// TIA Portal project "Sorting_Station_Project" (V16)
// Vorlageprojekt für das Buch mit Zielsystem S7-1200

(* hardware
DEVICE "S7-1200-Station_1"  S7-1200 Station
   slot 0: "Baugruppenträger_0"  Rack  V1.0
   slot 1: "PLC_1"  CPU 1211C DC/DC/DC  6ES7 211-1AE40-0XB0  V4.1
DEVICE "HMI_1"  KTP700 Basic PN
   slot 0: "HMI_1"  KTP700 Basic PN  6AV2 123-2GB03-0AX0  16.0.0.0
   slot 1: "HMI_RT_1"  KTP700 Basic PN  6AV2 123-2GB03-0AX0  16.0.0.0
   slot 5: "HMI_1.IE_CP_1"  PROFINET Interface  16.0.0.0
      slot 1: "PROFINET Interface_1"  PROFINET Interface
         slot 1: "Port_1"  Port
*)

// ===== PLC "PLC_1"  CPU 1211C DC/DC/DC =====

VAR_GLOBAL   // PLC tag table "Standard-Variablentabelle"
   "Entry_Conv_Stop" AT %M0.0 : Bool;
   "Entry_Conv" AT %Q0.1 : Bool;
   "Vision_Data" AT %ID30 : DInt;
   "nrig0" AT %M0.1 : Bool;
   "ntrig1" AT %M0.2 : Bool;
   "At_Exit_Sen" AT %I0.3 : Bool;
   "Exit_Conv" AT %Q0.2 : Bool;
   "ntrig2" AT %M0.3 : Bool;
   "Sorter_Memory" AT %MW2 : Int;
   "ntrig3" AT %M0.4 : Bool;
   "Sorter1B" AT %Q0.6 : Bool;
   "Sorter1T" AT %Q0.7 : Bool;
   "Sorter2B" AT %Q1.0 : Bool;
   "Sorter2T" AT %Q1.1 : Bool;
   "Sorter3B" AT %Q1.2 : Bool;
   "Sorter3T" AT %Q1.3 : Bool;
   "Start" AT %I0.0 : Bool;
   "Stop" AT %I0.1 : Bool;
   "System_Running" AT %M0.5 : Bool;
   "HMI_Start" AT %M0.6 : Bool;
   "HMI_Stop" AT %M0.7 : Bool;
   "Emergency" AT %I0.4 : Bool;
   "HMI_EM" AT %M1.0 : Bool;
   "Blue_lamp" AT %M1.1 : Bool;
   "Green_lamp" AT %M1.2 : Bool;
   "Silver_lamp" AT %M1.3 : Bool;
END_VAR

FUNCTION "MHJ-PLC-Lab-Function-S71200" : Void   // FC9000, SCL
{ S7_Optimized_Access := 'TRUE' }
VERSION : 0.1
   VAR_TEMP
      rdTimeReturn : Int;
      outputTime : DTL;
      SyncVal : Byte;
      forVal : Int;
      forVal_2 : Int;
      Value : Byte;
   END_VAR
   VAR CONSTANT
      CompVal : Byte := 16#34;
      Value_01 : Byte := 16#11;
      Value_01_DW : DWord := 16#A165_D992;
      Value_02_DW : DWord := 16#58BE_4401;
   END_VAR
BEGIN

   #Value:=PEEK(area := 16#82,
        dbNumber := 0,
        byteOffset := 511);
   #Value := #Value + 1;

   POKE(area := 16#82,
        dbNumber := 0,
        byteOffset := 511,
        value := #Value);

   POKE(area:=16#81,
        dbNumber:=0,
        byteOffset:=1016,
        value:=#Value_01_DW);
   POKE(area := 16#81,
        dbNumber := 0,
        byteOffset := 1020,
        value := #Value_02_DW);

   POKE(area := 16#81,
        dbNumber := 0,
        byteOffset := 511,
        value := B#16#00);

   FOR #forVal := 0 TO 120 DO
       FOR #forVal_2:=0 TO 10 DO
           #rdTimeReturn:=RD_SYS_T(#outputTime);
           #rdTimeReturn := WR_SYS_T(#outputTime);
           #rdTimeReturn := RD_SYS_T(#outputTime);
           #rdTimeReturn := WR_SYS_T(#outputTime);
       END_FOR;
       #SyncVal:= PEEK(area := 16#81,
                      dbNumber := 0,
                      byteOffset := 511);
       IF #SyncVal = #CompVal THEN
          GOTO M_1;
       END_IF;
   END_FOR;
   RETURN;

   M_1:
   POKE(area := 16#81,
        dbNumber := 0,
        byteOffset := 511,
        value := B#16#0);
END_FUNCTION

ORGANIZATION_BLOCK "Main"   // OB1, LAD, ProgramCycle
TITLE = "Main Program Sweep (Cycle)"
{ S7_Optimized_Access := 'TRUE' }
VERSION : 0.1
   VAR_INPUT
      Initial_Call : Bool;   // Initial call of this OB
      Remanence : Bool;   // =True, if remanent data are available
   END_VAR
   VAR_TEMP   // added for the SCL form of the ladder/FBD networks
      _w1 : Bool;
      _w2 : Bool;
      _w3 : Bool;
   END_VAR
BEGIN

REGION Network 1: Konnektierungsbaustein für PLC-Lab
   // Im Netzwerk 1 wird der Konnektierungsbaustein für PLC-Lab aufgerufen.
   // Dieser Aufruf darf nicht entfernt werden!
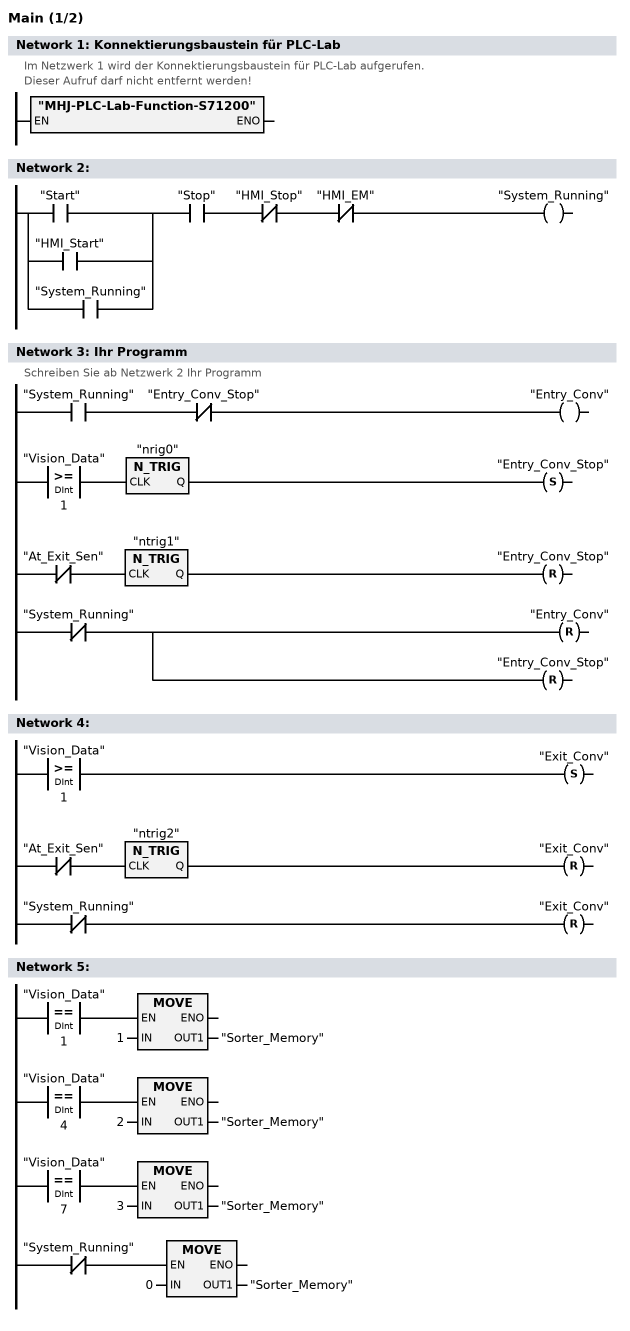
   RUNG wire#powerrail
      "MHJ-PLC-Lab-Function-S71200"()
   END_RUNG
   // the same network as SCL:
   "MHJ-PLC-Lab-Function-S71200"();
END_REGION

REGION Network 2
   RUNG wire#powerrail
      Contact( "Start" )
      wire#w1
      Contact( "Stop" )
      I_Contact( "HMI_Stop" )
      I_Contact( "HMI_EM" )
      Coil( "System_Running" )
   END_RUNG
   RUNG wire#powerrail
      Contact( "HMI_Start" )
   END_RUNG wire#w1
   RUNG wire#powerrail
      Contact( "System_Running" )
   END_RUNG wire#w1
   // the same network as SCL:
   "System_Running" := ("Start" OR "HMI_Start" OR "System_Running") AND "Stop" AND NOT "HMI_Stop" AND NOT "HMI_EM";
END_REGION

REGION Network 3: Ihr Programm
   // Schreiben Sie ab Netzwerk 2 Ihr Programm
   RUNG wire#powerrail
      Contact( "System_Running" )
      I_Contact( "Entry_Conv_Stop" )
      Coil( "Entry_Conv" )
   END_RUNG
   RUNG wire#powerrail
      { S7_Templates := "SrcType := DInt" } GE_Contact(in1 := "Vision_Data", in2 := 1)
      N_Trig( "nrig0" )
      S_Coil( "Entry_Conv_Stop" )
   END_RUNG
   RUNG wire#powerrail
      I_Contact( "At_Exit_Sen" )
      N_Trig( "ntrig1" )
      R_Coil( "Entry_Conv_Stop" )
   END_RUNG
   RUNG wire#powerrail
      I_Contact( "System_Running" )
      wire#w1
      R_Coil( "Entry_Conv" )
   END_RUNG
   RUNG wire#w1
      R_Coil( "Entry_Conv_Stop" )
   END_RUNG
   // the same network as SCL:
   "Entry_Conv" := "System_Running" AND NOT "Entry_Conv_Stop";
   #_w1 := "Vision_Data" >= 1;
   #_w2 := NOT #_w1 AND "nrig0";   // falling edge
   "nrig0" := #_w1;
   IF #_w2 THEN "Entry_Conv_Stop" := TRUE; END_IF;
   #_w3 := NOT (NOT "At_Exit_Sen") AND "ntrig1";   // falling edge
   "ntrig1" := NOT "At_Exit_Sen";
   IF #_w3 THEN "Entry_Conv_Stop" := FALSE; END_IF;
   IF NOT "System_Running" THEN
       "Entry_Conv" := FALSE;
       "Entry_Conv_Stop" := FALSE;
   END_IF;
END_REGION

REGION Network 4
   RUNG wire#powerrail
      { S7_Templates := "SrcType := DInt" } GE_Contact(in1 := "Vision_Data", in2 := 1)
      S_Coil( "Exit_Conv" )
   END_RUNG
   RUNG wire#powerrail
      I_Contact( "At_Exit_Sen" )
      N_Trig( "ntrig2" )
      R_Coil( "Exit_Conv" )
   END_RUNG
   RUNG wire#powerrail
      I_Contact( "System_Running" )
      R_Coil( "Exit_Conv" )
   END_RUNG
   // the same network as SCL:
   IF "Vision_Data" >= 1 THEN "Exit_Conv" := TRUE; END_IF;
   #_w1 := NOT (NOT "At_Exit_Sen") AND "ntrig2";   // falling edge
   "ntrig2" := NOT "At_Exit_Sen";
   IF #_w1 THEN "Exit_Conv" := FALSE; END_IF;
   IF NOT "System_Running" THEN "Exit_Conv" := FALSE; END_IF;
END_REGION

REGION Network 5
   RUNG wire#powerrail
      { S7_Templates := "SrcType := DInt" } EQ_Contact(in1 := "Vision_Data", in2 := 1)
      Move(in := 1, out1 => "Sorter_Memory")
   END_RUNG
   RUNG wire#powerrail
      { S7_Templates := "SrcType := DInt" } EQ_Contact(in1 := "Vision_Data", in2 := 4)
      Move(in := 2, out1 => "Sorter_Memory")
   END_RUNG
   RUNG wire#powerrail
      { S7_Templates := "SrcType := DInt" } EQ_Contact(in1 := "Vision_Data", in2 := 7)
      Move(in := 3, out1 => "Sorter_Memory")
   END_RUNG
   RUNG wire#powerrail
      I_Contact( "System_Running" )
      Move(in := 0, out1 => "Sorter_Memory")
   END_RUNG
   // the same network as SCL:
   IF "Vision_Data" = 1 THEN "Sorter_Memory" := 1; END_IF;
   IF "Vision_Data" = 4 THEN "Sorter_Memory" := 2; END_IF;
   IF "Vision_Data" = 7 THEN "Sorter_Memory" := 3; END_IF;
   IF NOT "System_Running" THEN "Sorter_Memory" := 0; END_IF;
END_REGION

REGION Network 6
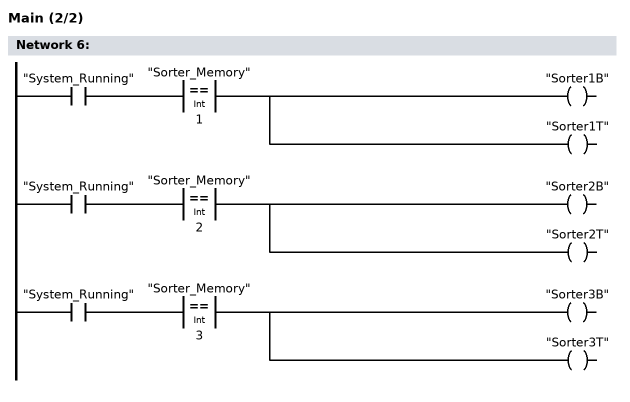
   RUNG wire#powerrail
      Contact( "System_Running" )
      { S7_Templates := "SrcType := Int" } EQ_Contact(in1 := "Sorter_Memory", in2 := 1)
      wire#w1
      Coil( "Sorter1B" )
   END_RUNG
   RUNG wire#w1
      Coil( "Sorter1T" )
   END_RUNG
   RUNG wire#powerrail
      Contact( "System_Running" )
      { S7_Templates := "SrcType := Int" } EQ_Contact(in1 := "Sorter_Memory", in2 := 2)
      wire#w2
      Coil( "Sorter2B" )
   END_RUNG
   RUNG wire#w2
      Coil( "Sorter2T" )
   END_RUNG
   RUNG wire#powerrail
      Contact( "System_Running" )
      { S7_Templates := "SrcType := Int" } EQ_Contact(in1 := "Sorter_Memory", in2 := 3)
      wire#w3
      Coil( "Sorter3B" )
   END_RUNG
   RUNG wire#w3
      Coil( "Sorter3T" )
   END_RUNG
   // the same network as SCL:
   "Sorter1B" := "System_Running" AND ("Sorter_Memory" = 1);
   "Sorter1T" := "Sorter1B";
   "Sorter2B" := "System_Running" AND ("Sorter_Memory" = 2);
   "Sorter2T" := "Sorter2B";
   "Sorter3B" := "System_Running" AND ("Sorter_Memory" = 3);
   "Sorter3T" := "Sorter3B";
END_REGION
END_ORGANIZATION_BLOCK

(* ===== HMI "HMI_RT_1" =====
system functions are stored by id; their names below are inferred from use
connection "HMI_Connection_1": ETHERNET, SMART_S7_1200_OMS

HMI tags "Default tag table"
   "Entry_Conv_Stop" : Bool = PLC Entry_Conv_Stop AT %M0.0, 100 ms
   "Entry_Conv" : Bool = PLC Entry_Conv AT %Q0.1, 100 ms
   "Vision_Data" : DInt = PLC Vision_Data AT %ID30, 100 ms
   "nrig0" : Bool = PLC nrig0 AT %M0.1, 100 ms
   "ntrig1" : Bool = PLC ntrig1 AT %M0.2, 100 ms
   "At_Exit_Sen" : Bool = PLC At_Exit_Sen AT %I0.3, 100 ms
   "Exit_Conv" : Bool = PLC Exit_Conv AT %Q0.2, 100 ms
   "ntrig2" : Bool = PLC ntrig2 AT %M0.3, 100 ms
   "Sorter_Memory" : Int = PLC Sorter_Memory AT %MW2, 100 ms
   "ntrig3" : Bool = PLC ntrig3 AT %M0.4, 100 ms
   "Sorter1B" : Bool = PLC Sorter1B AT %Q0.6, 100 ms
   "Sorter1T" : Bool = PLC Sorter1T AT %Q0.7, 100 ms
   "Sorter2B" : Bool = PLC Sorter2B AT %Q1.0, 100 ms
   "Sorter2T" : Bool = PLC Sorter2T AT %Q1.1, 100 ms
   "Sorter3B" : Bool = PLC Sorter3B AT %Q1.2, 100 ms
   "Sorter3T" : Bool = PLC Sorter3T AT %Q1.3, 100 ms
   "Start" : Bool = PLC Start AT %I0.0, 100 ms
   "Stop" : Bool = PLC Stop AT %I0.1, 100 ms
   "System_Running" : Bool = PLC System_Running AT %M0.5, 100 ms
   "Entry_Conv_Stop(1)" : Bool = PLC Entry_Conv_Stop AT %M0.0, 100 ms
   "Entry_Conv_Stop(2)" : Bool = PLC Entry_Conv_Stop AT %M0.0, 100 ms
   "HMI_Start" : Bool = PLC HMI_Start AT %M0.6, 100 ms
   "HMI_Stop" : Bool = PLC HMI_Stop AT %M0.7, 100 ms
   "Emergency" : Bool = PLC Emergency AT %I0.4, 100 ms
   "HMI_EM" : Bool = PLC HMI_EM AT %M1.0, 100 ms
   "Blue_lamp" : Bool = PLC Blue_lamp AT %M1.1, 100 ms
   "Green_lamp" : Bool = PLC Green_lamp AT %M1.2, 100 ms
   "Silver_lamp" : Bool = PLC Silver_lamp AT %M1.3, 100 ms

graphic list "Conveyor": 1 'Graphic_3'; 0 'Graphic_4'

screen "Main_Control_Screen" 800x480
   TextField "Text field_1" at 275,15 size 246x43; Text 'Sorting Station'
   Button "Button_1" at 23,262 size 96x32; TextOff 'Start'
      on Press: SetBit("HMI_Start")
      on Release: ResetBit("HMI_Start")
   Button "Button_2" at 147,262 size 96x32; TextOff 'Stop'
      on Press: SetBit("HMI_Stop")
      on Release: ResetBit("HMI_Stop")
   Circle "Circle_1" at 92,112 size 84x84
      Appearance <- "System_Running"
   TextField "Text field_2" at 66,208 size 121x23; Text 'System Status'
   TextField "Text field_4" at 482,126 size 129x23; Text 'Entry Conveyor'
   TextField "Text field_6" at 482,208 size 123x23; Text 'Exit Conveyor'
   Switch "Switch_1" at 23,322 size 220x44; CaptionText 'Switch'; TextOff 'Emergency OFF'; TextOn 'Emergency ON'
      ProcessValue <- "HMI_EM"
   Rectangle "Rectangle_1" at 628,201 size 79x36
      Appearance <- "Exit_Conv"
   Rectangle "Rectangle_2" at 628,120 size 79x36
      Appearance <- "Entry_Conv"
   TextField "Text field_3" at 356,309 size 193x23; Text 'Object Color Processed'
   Rectangle "Rectangle_3" at 572,300 size 52x25
      Appearance <- "Sorter1T"
   Rectangle "Rectangle_4" at 702,300 size 52x25
      Appearance <- "Sorter3T"
   Rectangle "Rectangle_5" at 639,300 size 52x25
      Appearance <- "Sorter2T"
   TextField "Text field_7" at 578,331 size 41x23; Text 'Blue'
   TextField "Text field_8" at 638,331 size 54x23; Text 'Green'
   TextField "Text field_9" at 703,331 size 51x23; Text 'Silver'
*)